FUNCTION_BLOCK G_buscar_numero
VAR_INPUT
	letra : STRING;
	cadena : STRING;
	
END_VAR
VAR_OUTPUT
	numero : REAL;
	error:BOOL;
END_VAR
VAR
	aux:INT;
	inicio:INT;
	espacio_siguiente:INT;
	cadena_recortada:STRING;
END_VAR

error:=FALSE;
numero:=0.99;
IF find(cadena,letra)=0 THEN
	error:=TRUE;
	ELSE
		aux:=find(cadena,letra);
		inicio:=aux + 1;
		cadena_recortada:=delete(cadena,aux,1);
		espacio_siguiente:=find(cadena_recortada,' ');
		IF espacio_siguiente=0 THEN
			espacio_siguiente := len(cadena_recortada)+1;
		END_IF
		numero:=STRING_TO_REAL(left(cadena_recortada,espacio_siguiente -1));
END_IF

END_FUNCTION_BLOCK

(* stored: Version 1.1.0.1, ProductVersion 3.1.4024.4
   POU G_buscar_numero: Id {86ea2a0f-187b-4f0f-bb18-001a1c7f87d7}, SpecialFunc None *)
